Fanuc KAREL source: kb00013.KL

-- PROVISIONAL review KL for V1013-1; original PC SHA256 d707eea87648146131c1fb6f80b5bdeb0938f956b17a5e35904925c6243d26da
-- Incomplete behavior may be omitted. Consult companion uncertainty JSON. Do not deploy.
PROGRAM KB00013
%NOLOCKGROUP
BEGIN
  -- UNRESOLVED_PC offsets 5-12; opcodes 9D,23
  -- UNRESOLVED_PC offsets 17-24; opcodes 9D,23
  -- UNRESOLVED_PC offsets 29-51; opcodes 27,22,22,22,31
  -- UNRESOLVED_PC offsets 56-60; opcodes 7F
END KB00013
